TYPE ST_EndStops :
STRUCT
END_STRUCT
END_TYPE

(* stored: Version 1.1.0.1, ProductVersion 3.1.4024.10
   DUT ST_EndStops: Id {9b48e6d4-525a-4647-a988-c36033c1d138} *)
